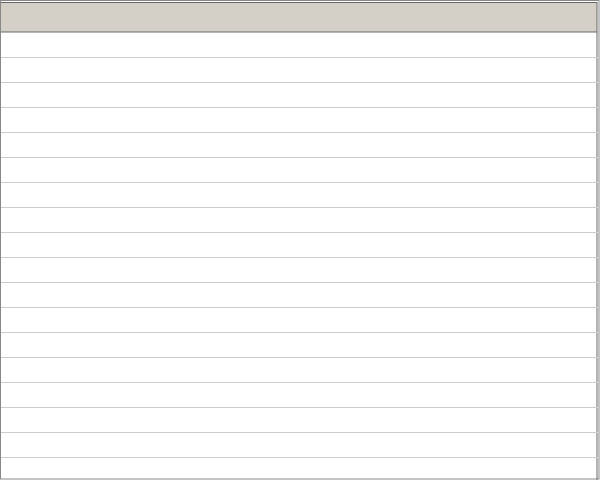
VISUALIZATION vEVENT_LOGGER  // 600x480
    Table (-3,2 600x480), data array: fbEventLogger.EventBuffer
        p3854506369: fbEventLogger.EventBuffer[INDEX].eEventType
        p1892666644: fbEventLogger.EventBuffer[INDEX].eEventSeverity
        p338671338: fbEventLogger.EventBuffer[INDEX].nEventIdentity
        p2170511999: fbEventLogger.EventBuffer[INDEX].sEventName
        p3723444502: fbEventLogger.EventBuffer[INDEX].sEventText
        p1218418051: fbEventLogger.EventBuffer[INDEX].dtTimestamp
END_VISUALIZATION

(* stored: Version 1.1.0.1, ProductVersion 3.1.4024.12
   Visu vEVENT_LOGGER: Id {4d490072-8c68-4228-b815-8b8173235622} *)
